# EPICS IOC start-up script: iocsh/ethercatmcEL1252-OneChannel.iocsh
ethercatmcCreateAsynParam $(MOTOR_PORT) UTCEL1252P Int64
ethercatmcCreateAsynParam $(MOTOR_PORT) UTCEL1252N Int64

dbLoadRecords("ethercatmcEL1252-OneChannel.template", "P=$(P), R=$(R), MOTOR_PORT=$(MOTOR_PORT), CHNO=$(CHNO)")
